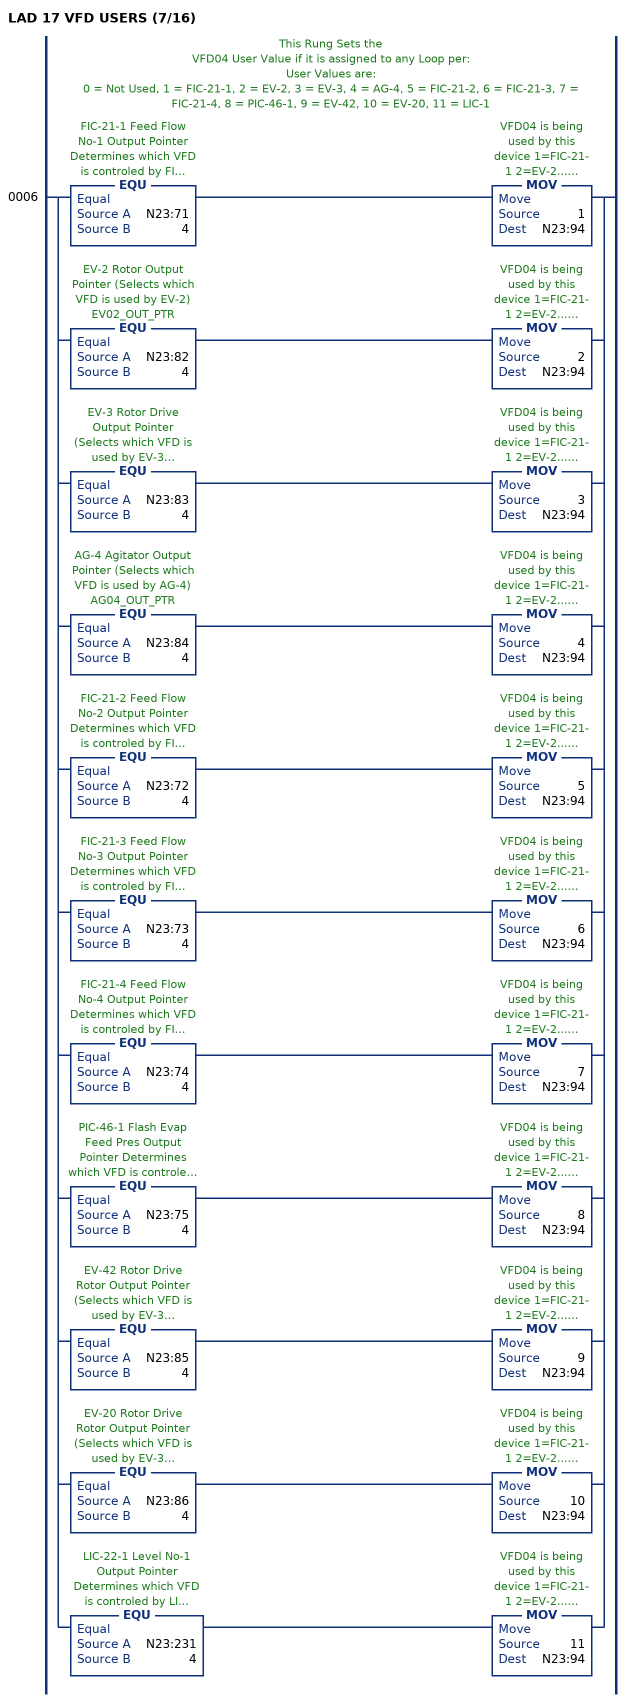
% Rung: 6 %
% This Rung Sets the
% VFD04 User Value if it is assigned to any Loop per:
% 
% User Values are:
% 0 = Not Used, 1 = FIC-21-1, 2 = EV-2, 3 = EV-3, 4 = AG-4, 5 = FIC-21-2, 6 = FIC-21-3, 7 = FIC-21-4, 8 = PIC-46-1, 9 = EV-42, 10 = EV-20, 11 = LIC-1 %
SOR BST EQU N23:71 4 MOV 1 N23:94 NXB EQU N23:82 4 MOV 2 N23:94 NXB EQU N23:83 4 MOV 3 N23:94 NXB EQU N23:84 4 MOV 4 N23:94 NXB EQU N23:72 4 MOV 5 N23:94 NXB EQU N23:73 4 MOV 6 N23:94 NXB EQU N23:74 4 MOV 7 N23:94 NXB EQU N23:75 4 MOV 8 N23:94 NXB EQU N23:85 4 MOV 9 N23:94 NXB EQU N23:86 4 MOV 10 N23:94 NXB EQU N23:231 4 MOV 11 N23:94 BND EOR
%   N23:71  FIC211_OUT_PTR  "FIC-21-1 Feed Flow No-1 Output Pointer Determines which VFD is controled by FIC" %
%   N23:94  VFD04_USER  "VFD04 is being used by this device 1=FIC-21-1 2=EV-2...." %
%   N23:82  EV02_OUT_PTR  "EV-2 Rotor Output Pointer (Selects which VFD is used by EV-2)" %
%   N23:83  EV03_OUT_PTR  "EV-3 Rotor Drive Output Pointer (Selects which VFD is used by EV-3)" %
%   N23:84  AG04_OUT_PTR  "AG-4 Agitator Output Pointer (Selects which VFD is used by AG-4)" %
%   N23:72  FIC212_OUT_PTR  "FIC-21-2 Feed Flow No-2 Output Pointer Determines which VFD is controled by FIC" %
%   N23:73  FIC213_OUT_PTR  "FIC-21-3 Feed Flow No-3 Output Pointer Determines which VFD is controled by FIC" %
%   N23:74  FIC214_OUT_PTR  "FIC-21-4 Feed Flow No-4 Output Pointer Determines which VFD is controled by FIC" %
%   N23:75  PIC461_OUT_PTR  "PIC-46-1 Flash Evap Feed Pres Output Pointer Determines which VFD is controled by FIC" %
%   N23:85  EV42_OUT_PTR  "EV-42 Rotor Drive Rotor Output Pointer (Selects which VFD is used by EV-3)" %
%   N23:86  EV20_OUT_PTR  "EV-20 Rotor Drive Rotor Output Pointer (Selects which VFD is used by EV-3)" %
%   N23:231  LIC221_OUT_PTR  "LIC-22-1 Level No-1 Output Pointer Determines which VFD is controled by LIC" %

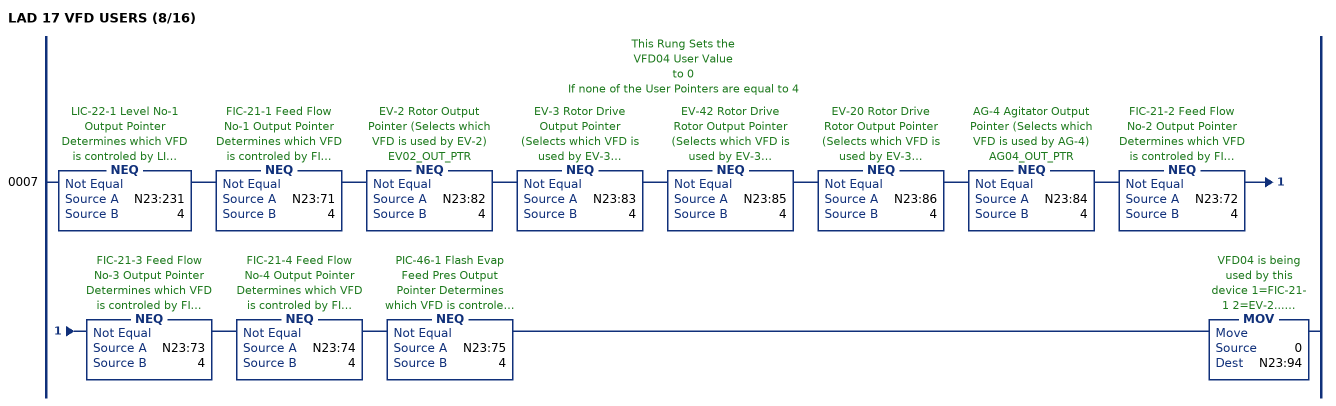
% Rung: 7 %
% This Rung Sets the
% VFD04 User Value
% to 0
% If none of the User Pointers are equal to 4 %
SOR NEQ N23:231 4 NEQ N23:71 4 NEQ N23:82 4 NEQ N23:83 4 NEQ N23:85 4 NEQ N23:86 4 NEQ N23:84 4 NEQ N23:72 4 NEQ N23:73 4 NEQ N23:74 4 NEQ N23:75 4 MOV 0 N23:94 EOR
%   N23:231  LIC221_OUT_PTR  "LIC-22-1 Level No-1 Output Pointer Determines which VFD is controled by LIC" %
%   N23:71  FIC211_OUT_PTR  "FIC-21-1 Feed Flow No-1 Output Pointer Determines which VFD is controled by FIC" %
%   N23:82  EV02_OUT_PTR  "EV-2 Rotor Output Pointer (Selects which VFD is used by EV-2)" %
%   N23:83  EV03_OUT_PTR  "EV-3 Rotor Drive Output Pointer (Selects which VFD is used by EV-3)" %
%   N23:85  EV42_OUT_PTR  "EV-42 Rotor Drive Rotor Output Pointer (Selects which VFD is used by EV-3)" %
%   N23:86  EV20_OUT_PTR  "EV-20 Rotor Drive Rotor Output Pointer (Selects which VFD is used by EV-3)" %
%   N23:84  AG04_OUT_PTR  "AG-4 Agitator Output Pointer (Selects which VFD is used by AG-4)" %
%   N23:72  FIC212_OUT_PTR  "FIC-21-2 Feed Flow No-2 Output Pointer Determines which VFD is controled by FIC" %
%   N23:73  FIC213_OUT_PTR  "FIC-21-3 Feed Flow No-3 Output Pointer Determines which VFD is controled by FIC" %
%   N23:74  FIC214_OUT_PTR  "FIC-21-4 Feed Flow No-4 Output Pointer Determines which VFD is controled by FIC" %
%   N23:75  PIC461_OUT_PTR  "PIC-46-1 Flash Evap Feed Pres Output Pointer Determines which VFD is controled by FIC" %
%   N23:94  VFD04_USER  "VFD04 is being used by this device 1=FIC-21-1 2=EV-2...." %

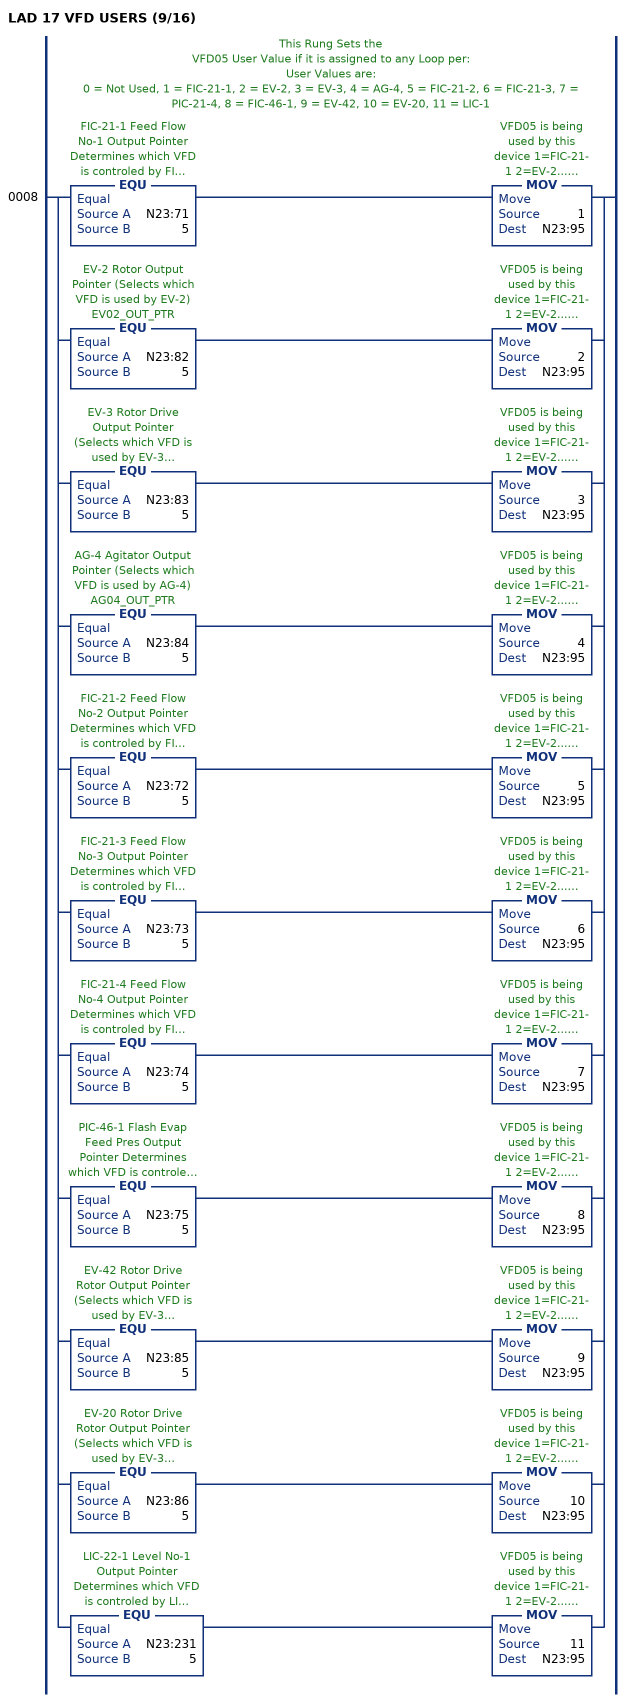
% Rung: 8 %
% This Rung Sets the
% VFD05 User Value if it is assigned to any Loop per:
% 
% User Values are:
% 0 = Not Used, 1 = FIC-21-1, 2 = EV-2, 3 = EV-3, 4 = AG-4, 5 = FIC-21-2, 6 = FIC-21-3, 7 = PIC-21-4, 8 = FIC-46-1, 9 = EV-42, 10 = EV-20, 11 = LIC-1 %
SOR BST EQU N23:71 5 MOV 1 N23:95 NXB EQU N23:82 5 MOV 2 N23:95 NXB EQU N23:83 5 MOV 3 N23:95 NXB EQU N23:84 5 MOV 4 N23:95 NXB EQU N23:72 5 MOV 5 N23:95 NXB EQU N23:73 5 MOV 6 N23:95 NXB EQU N23:74 5 MOV 7 N23:95 NXB EQU N23:75 5 MOV 8 N23:95 NXB EQU N23:85 5 MOV 9 N23:95 NXB EQU N23:86 5 MOV 10 N23:95 NXB EQU N23:231 5 MOV 11 N23:95 BND EOR
%   N23:71  FIC211_OUT_PTR  "FIC-21-1 Feed Flow No-1 Output Pointer Determines which VFD is controled by FIC" %
%   N23:95  VFD05_USER  "VFD05 is being used by this device 1=FIC-21-1 2=EV-2...." %
%   N23:82  EV02_OUT_PTR  "EV-2 Rotor Output Pointer (Selects which VFD is used by EV-2)" %
%   N23:83  EV03_OUT_PTR  "EV-3 Rotor Drive Output Pointer (Selects which VFD is used by EV-3)" %
%   N23:84  AG04_OUT_PTR  "AG-4 Agitator Output Pointer (Selects which VFD is used by AG-4)" %
%   N23:72  FIC212_OUT_PTR  "FIC-21-2 Feed Flow No-2 Output Pointer Determines which VFD is controled by FIC" %
%   N23:73  FIC213_OUT_PTR  "FIC-21-3 Feed Flow No-3 Output Pointer Determines which VFD is controled by FIC" %
%   N23:74  FIC214_OUT_PTR  "FIC-21-4 Feed Flow No-4 Output Pointer Determines which VFD is controled by FIC" %
%   N23:75  PIC461_OUT_PTR  "PIC-46-1 Flash Evap Feed Pres Output Pointer Determines which VFD is controled by FIC" %
%   N23:85  EV42_OUT_PTR  "EV-42 Rotor Drive Rotor Output Pointer (Selects which VFD is used by EV-3)" %
%   N23:86  EV20_OUT_PTR  "EV-20 Rotor Drive Rotor Output Pointer (Selects which VFD is used by EV-3)" %
%   N23:231  LIC221_OUT_PTR  "LIC-22-1 Level No-1 Output Pointer Determines which VFD is controled by LIC" %

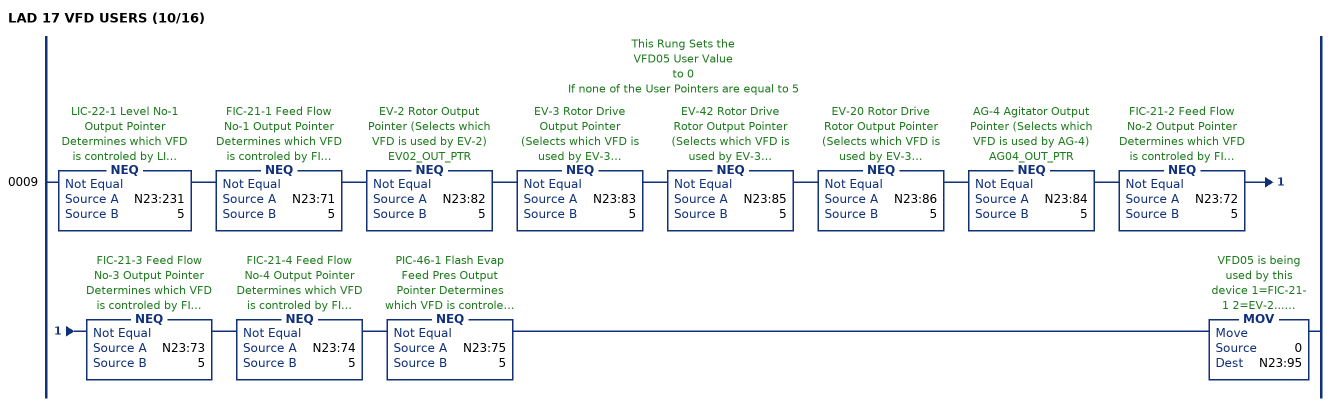
% Rung: 9 %
% This Rung Sets the
% VFD05 User Value
% to 0
% If none of the User Pointers are equal to 5 %
SOR NEQ N23:231 5 NEQ N23:71 5 NEQ N23:82 5 NEQ N23:83 5 NEQ N23:85 5 NEQ N23:86 5 NEQ N23:84 5 NEQ N23:72 5 NEQ N23:73 5 NEQ N23:74 5 NEQ N23:75 5 MOV 0 N23:95 EOR
%   N23:231  LIC221_OUT_PTR  "LIC-22-1 Level No-1 Output Pointer Determines which VFD is controled by LIC" %
%   N23:71  FIC211_OUT_PTR  "FIC-21-1 Feed Flow No-1 Output Pointer Determines which VFD is controled by FIC" %
%   N23:82  EV02_OUT_PTR  "EV-2 Rotor Output Pointer (Selects which VFD is used by EV-2)" %
%   N23:83  EV03_OUT_PTR  "EV-3 Rotor Drive Output Pointer (Selects which VFD is used by EV-3)" %
%   N23:85  EV42_OUT_PTR  "EV-42 Rotor Drive Rotor Output Pointer (Selects which VFD is used by EV-3)" %
%   N23:86  EV20_OUT_PTR  "EV-20 Rotor Drive Rotor Output Pointer (Selects which VFD is used by EV-3)" %
%   N23:84  AG04_OUT_PTR  "AG-4 Agitator Output Pointer (Selects which VFD is used by AG-4)" %
%   N23:72  FIC212_OUT_PTR  "FIC-21-2 Feed Flow No-2 Output Pointer Determines which VFD is controled by FIC" %
%   N23:73  FIC213_OUT_PTR  "FIC-21-3 Feed Flow No-3 Output Pointer Determines which VFD is controled by FIC" %
%   N23:74  FIC214_OUT_PTR  "FIC-21-4 Feed Flow No-4 Output Pointer Determines which VFD is controled by FIC" %
%   N23:75  PIC461_OUT_PTR  "PIC-46-1 Flash Evap Feed Pres Output Pointer Determines which VFD is controled by FIC" %
%   N23:95  VFD05_USER  "VFD05 is being used by this device 1=FIC-21-1 2=EV-2...." %

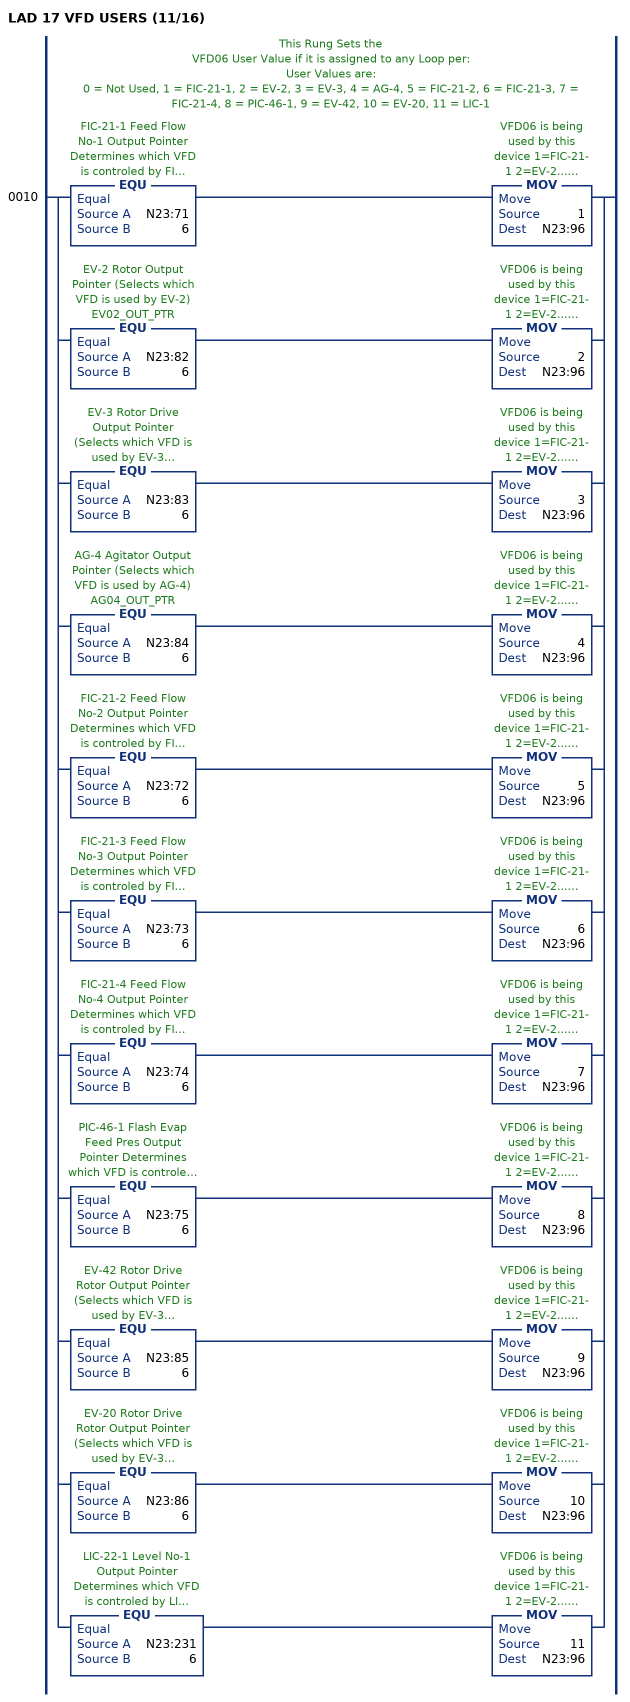
% Rung: 10 %
% This Rung Sets the
% VFD06 User Value if it is assigned to any Loop per:
% 
% User Values are:
% 0 = Not Used, 1 = FIC-21-1, 2 = EV-2, 3 = EV-3, 4 = AG-4, 5 = FIC-21-2, 6 = FIC-21-3, 7 = FIC-21-4, 8 = PIC-46-1, 9 = EV-42, 10 = EV-20, 11 = LIC-1 %
SOR BST EQU N23:71 6 MOV 1 N23:96 NXB EQU N23:82 6 MOV 2 N23:96 NXB EQU N23:83 6 MOV 3 N23:96 NXB EQU N23:84 6 MOV 4 N23:96 NXB EQU N23:72 6 MOV 5 N23:96 NXB EQU N23:73 6 MOV 6 N23:96 NXB EQU N23:74 6 MOV 7 N23:96 NXB EQU N23:75 6 MOV 8 N23:96 NXB EQU N23:85 6 MOV 9 N23:96 NXB EQU N23:86 6 MOV 10 N23:96 NXB EQU N23:231 6 MOV 11 N23:96 BND EOR
%   N23:71  FIC211_OUT_PTR  "FIC-21-1 Feed Flow No-1 Output Pointer Determines which VFD is controled by FIC" %
%   N23:96  VFD06_USER  "VFD06 is being used by this device 1=FIC-21-1 2=EV-2...." %
%   N23:82  EV02_OUT_PTR  "EV-2 Rotor Output Pointer (Selects which VFD is used by EV-2)" %
%   N23:83  EV03_OUT_PTR  "EV-3 Rotor Drive Output Pointer (Selects which VFD is used by EV-3)" %
%   N23:84  AG04_OUT_PTR  "AG-4 Agitator Output Pointer (Selects which VFD is used by AG-4)" %
%   N23:72  FIC212_OUT_PTR  "FIC-21-2 Feed Flow No-2 Output Pointer Determines which VFD is controled by FIC" %
%   N23:73  FIC213_OUT_PTR  "FIC-21-3 Feed Flow No-3 Output Pointer Determines which VFD is controled by FIC" %
%   N23:74  FIC214_OUT_PTR  "FIC-21-4 Feed Flow No-4 Output Pointer Determines which VFD is controled by FIC" %
%   N23:75  PIC461_OUT_PTR  "PIC-46-1 Flash Evap Feed Pres Output Pointer Determines which VFD is controled by FIC" %
%   N23:85  EV42_OUT_PTR  "EV-42 Rotor Drive Rotor Output Pointer (Selects which VFD is used by EV-3)" %
%   N23:86  EV20_OUT_PTR  "EV-20 Rotor Drive Rotor Output Pointer (Selects which VFD is used by EV-3)" %
%   N23:231  LIC221_OUT_PTR  "LIC-22-1 Level No-1 Output Pointer Determines which VFD is controled by LIC" %

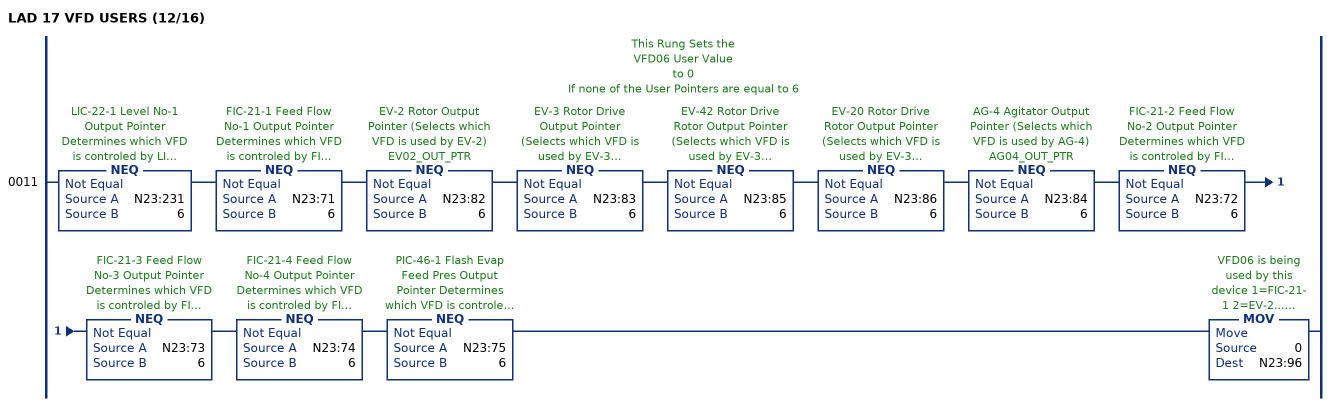
% Rung: 11 %
% This Rung Sets the
% VFD06 User Value
% to 0
% If none of the User Pointers are equal to 6 %
SOR NEQ N23:231 6 NEQ N23:71 6 NEQ N23:82 6 NEQ N23:83 6 NEQ N23:85 6 NEQ N23:86 6 NEQ N23:84 6 NEQ N23:72 6 NEQ N23:73 6 NEQ N23:74 6 NEQ N23:75 6 MOV 0 N23:96 EOR
%   N23:231  LIC221_OUT_PTR  "LIC-22-1 Level No-1 Output Pointer Determines which VFD is controled by LIC" %
%   N23:71  FIC211_OUT_PTR  "FIC-21-1 Feed Flow No-1 Output Pointer Determines which VFD is controled by FIC" %
%   N23:82  EV02_OUT_PTR  "EV-2 Rotor Output Pointer (Selects which VFD is used by EV-2)" %
%   N23:83  EV03_OUT_PTR  "EV-3 Rotor Drive Output Pointer (Selects which VFD is used by EV-3)" %
%   N23:85  EV42_OUT_PTR  "EV-42 Rotor Drive Rotor Output Pointer (Selects which VFD is used by EV-3)" %
%   N23:86  EV20_OUT_PTR  "EV-20 Rotor Drive Rotor Output Pointer (Selects which VFD is used by EV-3)" %
%   N23:84  AG04_OUT_PTR  "AG-4 Agitator Output Pointer (Selects which VFD is used by AG-4)" %
%   N23:72  FIC212_OUT_PTR  "FIC-21-2 Feed Flow No-2 Output Pointer Determines which VFD is controled by FIC" %
%   N23:73  FIC213_OUT_PTR  "FIC-21-3 Feed Flow No-3 Output Pointer Determines which VFD is controled by FIC" %
%   N23:74  FIC214_OUT_PTR  "FIC-21-4 Feed Flow No-4 Output Pointer Determines which VFD is controled by FIC" %
%   N23:75  PIC461_OUT_PTR  "PIC-46-1 Flash Evap Feed Pres Output Pointer Determines which VFD is controled by FIC" %
%   N23:96  VFD06_USER  "VFD06 is being used by this device 1=FIC-21-1 2=EV-2...." %

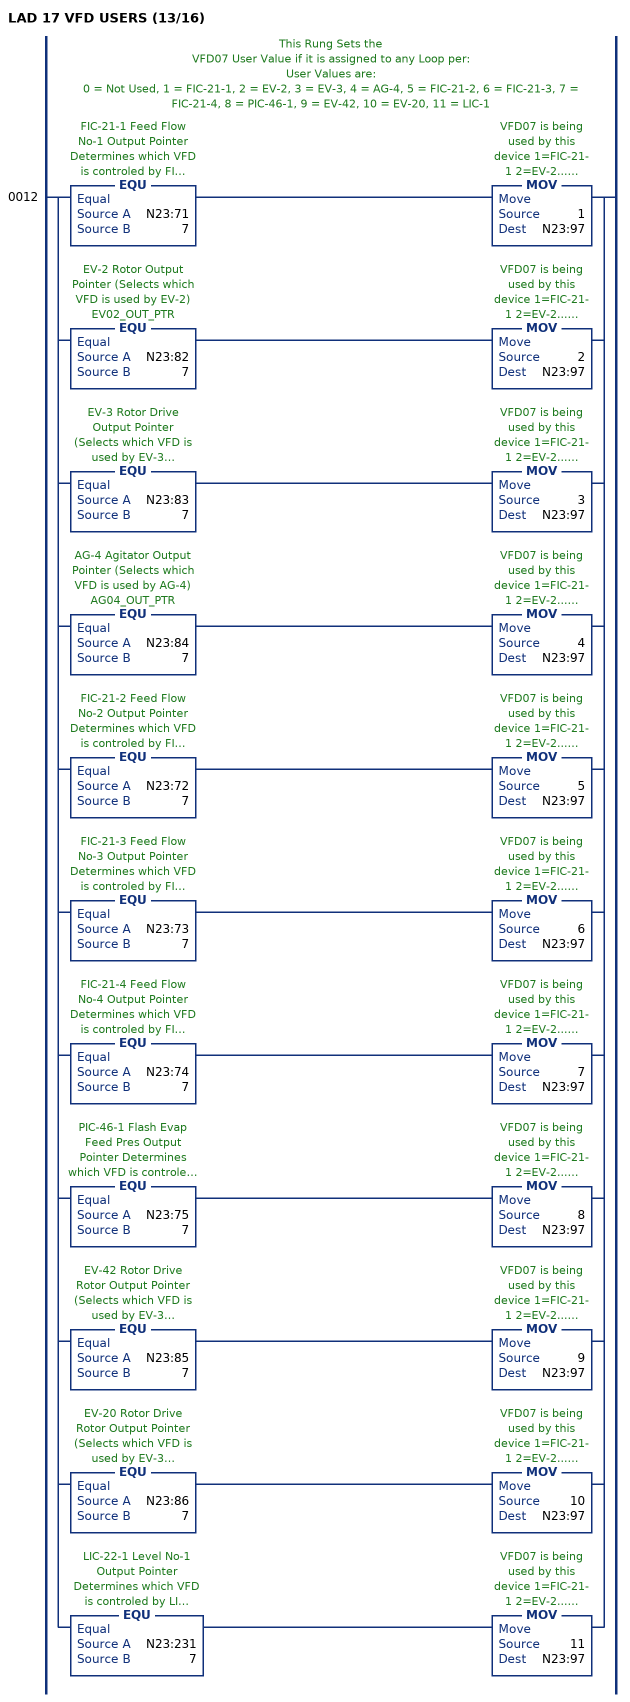
% Rung: 12 %
% This Rung Sets the
% VFD07 User Value if it is assigned to any Loop per:
% 
% User Values are:
% 0 = Not Used, 1 = FIC-21-1, 2 = EV-2, 3 = EV-3, 4 = AG-4, 5 = FIC-21-2, 6 = FIC-21-3, 7 = FIC-21-4, 8 = PIC-46-1, 9 = EV-42, 10 = EV-20, 11 = LIC-1 %
SOR BST EQU N23:71 7 MOV 1 N23:97 NXB EQU N23:82 7 MOV 2 N23:97 NXB EQU N23:83 7 MOV 3 N23:97 NXB EQU N23:84 7 MOV 4 N23:97 NXB EQU N23:72 7 MOV 5 N23:97 NXB EQU N23:73 7 MOV 6 N23:97 NXB EQU N23:74 7 MOV 7 N23:97 NXB EQU N23:75 7 MOV 8 N23:97 NXB EQU N23:85 7 MOV 9 N23:97 NXB EQU N23:86 7 MOV 10 N23:97 NXB EQU N23:231 7 MOV 11 N23:97 BND EOR
%   N23:71  FIC211_OUT_PTR  "FIC-21-1 Feed Flow No-1 Output Pointer Determines which VFD is controled by FIC" %
%   N23:97  VFD07_USER  "VFD07 is being used by this device 1=FIC-21-1 2=EV-2...." %
%   N23:82  EV02_OUT_PTR  "EV-2 Rotor Output Pointer (Selects which VFD is used by EV-2)" %
%   N23:83  EV03_OUT_PTR  "EV-3 Rotor Drive Output Pointer (Selects which VFD is used by EV-3)" %
%   N23:84  AG04_OUT_PTR  "AG-4 Agitator Output Pointer (Selects which VFD is used by AG-4)" %
%   N23:72  FIC212_OUT_PTR  "FIC-21-2 Feed Flow No-2 Output Pointer Determines which VFD is controled by FIC" %
%   N23:73  FIC213_OUT_PTR  "FIC-21-3 Feed Flow No-3 Output Pointer Determines which VFD is controled by FIC" %
%   N23:74  FIC214_OUT_PTR  "FIC-21-4 Feed Flow No-4 Output Pointer Determines which VFD is controled by FIC" %
%   N23:75  PIC461_OUT_PTR  "PIC-46-1 Flash Evap Feed Pres Output Pointer Determines which VFD is controled by FIC" %
%   N23:85  EV42_OUT_PTR  "EV-42 Rotor Drive Rotor Output Pointer (Selects which VFD is used by EV-3)" %
%   N23:86  EV20_OUT_PTR  "EV-20 Rotor Drive Rotor Output Pointer (Selects which VFD is used by EV-3)" %
%   N23:231  LIC221_OUT_PTR  "LIC-22-1 Level No-1 Output Pointer Determines which VFD is controled by LIC" %

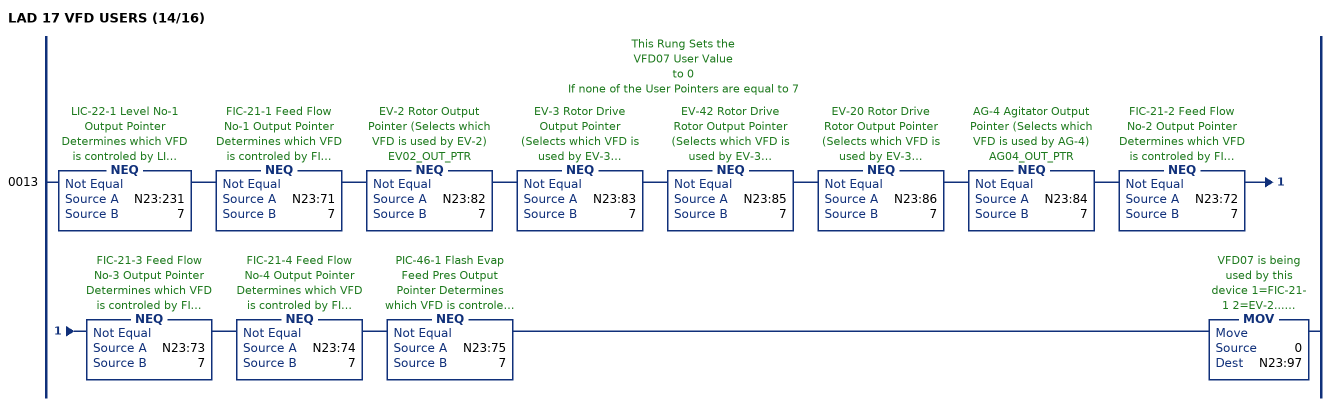
% Rung: 13 %
% This Rung Sets the
% VFD07 User Value
% to 0
% If none of the User Pointers are equal to 7 %
SOR NEQ N23:231 7 NEQ N23:71 7 NEQ N23:82 7 NEQ N23:83 7 NEQ N23:85 7 NEQ N23:86 7 NEQ N23:84 7 NEQ N23:72 7 NEQ N23:73 7 NEQ N23:74 7 NEQ N23:75 7 MOV 0 N23:97 EOR
%   N23:231  LIC221_OUT_PTR  "LIC-22-1 Level No-1 Output Pointer Determines which VFD is controled by LIC" %
%   N23:71  FIC211_OUT_PTR  "FIC-21-1 Feed Flow No-1 Output Pointer Determines which VFD is controled by FIC" %
%   N23:82  EV02_OUT_PTR  "EV-2 Rotor Output Pointer (Selects which VFD is used by EV-2)" %
%   N23:83  EV03_OUT_PTR  "EV-3 Rotor Drive Output Pointer (Selects which VFD is used by EV-3)" %
%   N23:85  EV42_OUT_PTR  "EV-42 Rotor Drive Rotor Output Pointer (Selects which VFD is used by EV-3)" %
%   N23:86  EV20_OUT_PTR  "EV-20 Rotor Drive Rotor Output Pointer (Selects which VFD is used by EV-3)" %
%   N23:84  AG04_OUT_PTR  "AG-4 Agitator Output Pointer (Selects which VFD is used by AG-4)" %
%   N23:72  FIC212_OUT_PTR  "FIC-21-2 Feed Flow No-2 Output Pointer Determines which VFD is controled by FIC" %
%   N23:73  FIC213_OUT_PTR  "FIC-21-3 Feed Flow No-3 Output Pointer Determines which VFD is controled by FIC" %
%   N23:74  FIC214_OUT_PTR  "FIC-21-4 Feed Flow No-4 Output Pointer Determines which VFD is controled by FIC" %
%   N23:75  PIC461_OUT_PTR  "PIC-46-1 Flash Evap Feed Pres Output Pointer Determines which VFD is controled by FIC" %
%   N23:97  VFD07_USER  "VFD07 is being used by this device 1=FIC-21-1 2=EV-2...." %

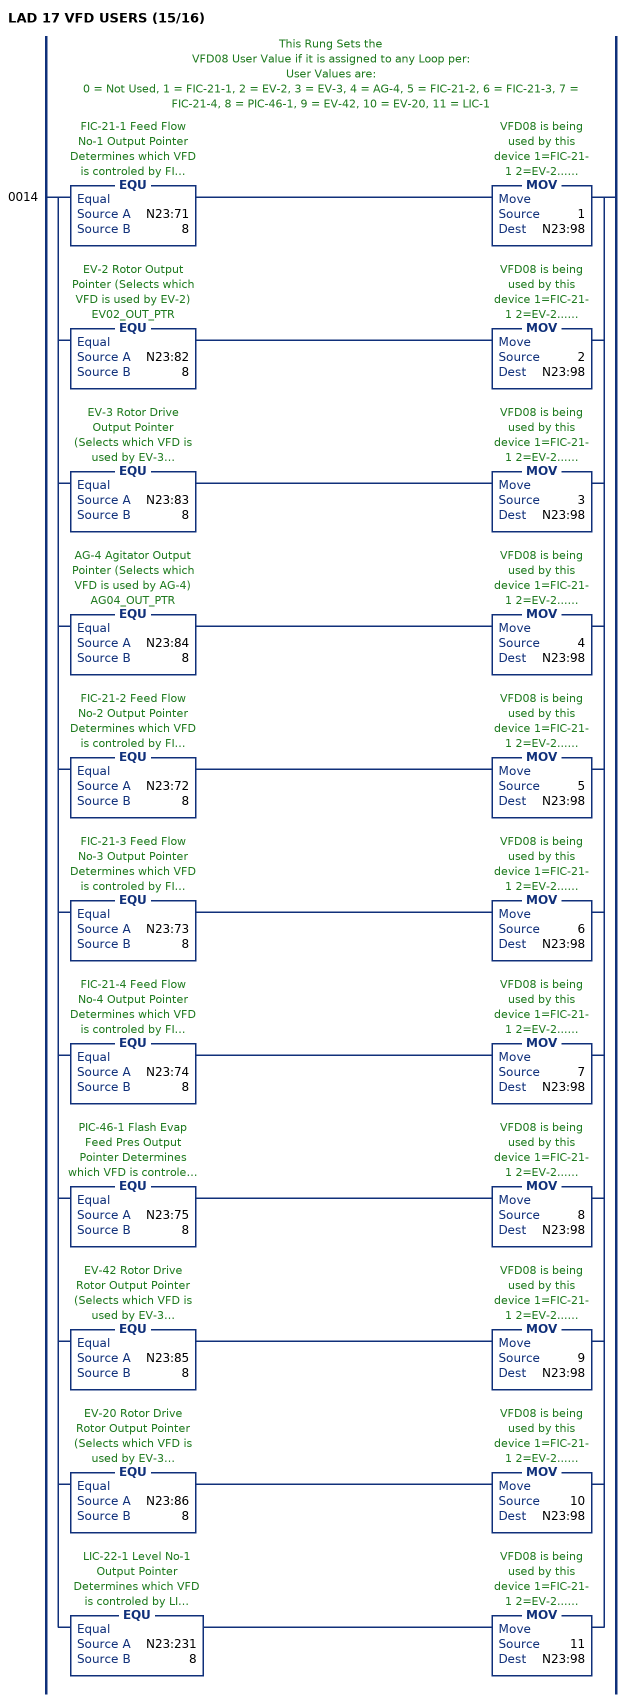
% Rung: 14 %
% This Rung Sets the
% VFD08 User Value if it is assigned to any Loop per:
% 
% User Values are:
% 0 = Not Used, 1 = FIC-21-1, 2 = EV-2, 3 = EV-3, 4 = AG-4, 5 = FIC-21-2, 6 = FIC-21-3, 7 = FIC-21-4, 8 = PIC-46-1, 9 = EV-42, 10 = EV-20, 11 = LIC-1 %
SOR BST EQU N23:71 8 MOV 1 N23:98 NXB EQU N23:82 8 MOV 2 N23:98 NXB EQU N23:83 8 MOV 3 N23:98 NXB EQU N23:84 8 MOV 4 N23:98 NXB EQU N23:72 8 MOV 5 N23:98 NXB EQU N23:73 8 MOV 6 N23:98 NXB EQU N23:74 8 MOV 7 N23:98 NXB EQU N23:75 8 MOV 8 N23:98 NXB EQU N23:85 8 MOV 9 N23:98 NXB EQU N23:86 8 MOV 10 N23:98 NXB EQU N23:231 8 MOV 11 N23:98 BND EOR
%   N23:71  FIC211_OUT_PTR  "FIC-21-1 Feed Flow No-1 Output Pointer Determines which VFD is controled by FIC" %
%   N23:98  VFD08_USER  "VFD08 is being used by this device 1=FIC-21-1 2=EV-2...." %
%   N23:82  EV02_OUT_PTR  "EV-2 Rotor Output Pointer (Selects which VFD is used by EV-2)" %
%   N23:83  EV03_OUT_PTR  "EV-3 Rotor Drive Output Pointer (Selects which VFD is used by EV-3)" %
%   N23:84  AG04_OUT_PTR  "AG-4 Agitator Output Pointer (Selects which VFD is used by AG-4)" %
%   N23:72  FIC212_OUT_PTR  "FIC-21-2 Feed Flow No-2 Output Pointer Determines which VFD is controled by FIC" %
%   N23:73  FIC213_OUT_PTR  "FIC-21-3 Feed Flow No-3 Output Pointer Determines which VFD is controled by FIC" %
%   N23:74  FIC214_OUT_PTR  "FIC-21-4 Feed Flow No-4 Output Pointer Determines which VFD is controled by FIC" %
%   N23:75  PIC461_OUT_PTR  "PIC-46-1 Flash Evap Feed Pres Output Pointer Determines which VFD is controled by FIC" %
%   N23:85  EV42_OUT_PTR  "EV-42 Rotor Drive Rotor Output Pointer (Selects which VFD is used by EV-3)" %
%   N23:86  EV20_OUT_PTR  "EV-20 Rotor Drive Rotor Output Pointer (Selects which VFD is used by EV-3)" %
%   N23:231  LIC221_OUT_PTR  "LIC-22-1 Level No-1 Output Pointer Determines which VFD is controled by LIC" %

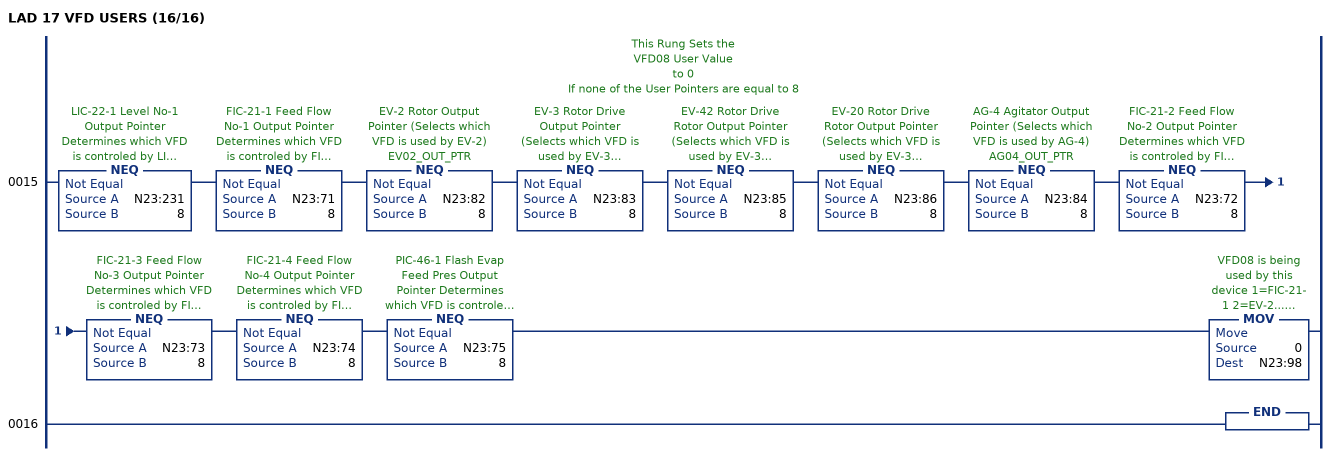
% Rung: 15 %
% This Rung Sets the
% VFD08 User Value
% to 0
% If none of the User Pointers are equal to 8 %
SOR NEQ N23:231 8 NEQ N23:71 8 NEQ N23:82 8 NEQ N23:83 8 NEQ N23:85 8 NEQ N23:86 8 NEQ N23:84 8 NEQ N23:72 8 NEQ N23:73 8 NEQ N23:74 8 NEQ N23:75 8 MOV 0 N23:98 EOR
%   N23:231  LIC221_OUT_PTR  "LIC-22-1 Level No-1 Output Pointer Determines which VFD is controled by LIC" %
%   N23:71  FIC211_OUT_PTR  "FIC-21-1 Feed Flow No-1 Output Pointer Determines which VFD is controled by FIC" %
%   N23:82  EV02_OUT_PTR  "EV-2 Rotor Output Pointer (Selects which VFD is used by EV-2)" %
%   N23:83  EV03_OUT_PTR  "EV-3 Rotor Drive Output Pointer (Selects which VFD is used by EV-3)" %
%   N23:85  EV42_OUT_PTR  "EV-42 Rotor Drive Rotor Output Pointer (Selects which VFD is used by EV-3)" %
%   N23:86  EV20_OUT_PTR  "EV-20 Rotor Drive Rotor Output Pointer (Selects which VFD is used by EV-3)" %
%   N23:84  AG04_OUT_PTR  "AG-4 Agitator Output Pointer (Selects which VFD is used by AG-4)" %
%   N23:72  FIC212_OUT_PTR  "FIC-21-2 Feed Flow No-2 Output Pointer Determines which VFD is controled by FIC" %
%   N23:73  FIC213_OUT_PTR  "FIC-21-3 Feed Flow No-3 Output Pointer Determines which VFD is controled by FIC" %
%   N23:74  FIC214_OUT_PTR  "FIC-21-4 Feed Flow No-4 Output Pointer Determines which VFD is controled by FIC" %
%   N23:75  PIC461_OUT_PTR  "PIC-46-1 Flash Evap Feed Pres Output Pointer Determines which VFD is controled by FIC" %
%   N23:98  VFD08_USER  "VFD08 is being used by this device 1=FIC-21-1 2=EV-2...." %
% Rung: 16 %
SOR END EOR

LADDER 31 "MOVE TES"    % Move TE Info to Sequencial Locations, etc %
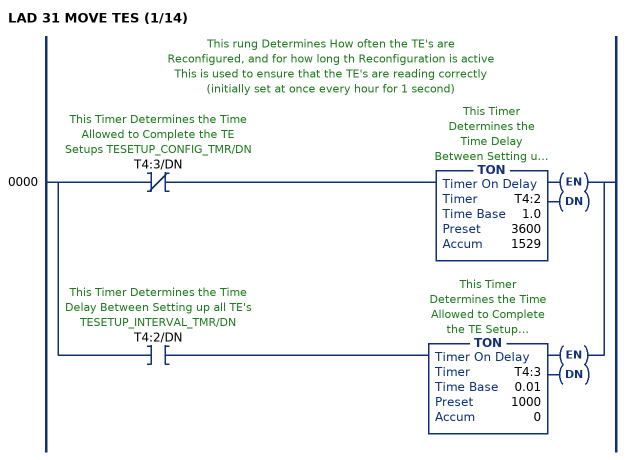
% Rung: 0 %
% This rung Determines How often the TE's are
% Reconfigured, and for how long th Reconfiguration is active
% This is used to ensure that the TE's are reading correctly
%    (initially set at once every hour for 1 second) %
SOR BST XIO T4:3/DN TON T4:2 1.0 3600 1529 NXB XIC T4:2/DN TON T4:3 0.01 1000 0 BND EOR
%   T4:3  TESETUP_CONFIG_TMR  "This Timer Determines the Time Allowed to Complete the TE Setups" %
%   T4:2  TESETUP_INTERVAL_TMR  "This Timer Determines the Time Delay Between Setting up all TE's" %

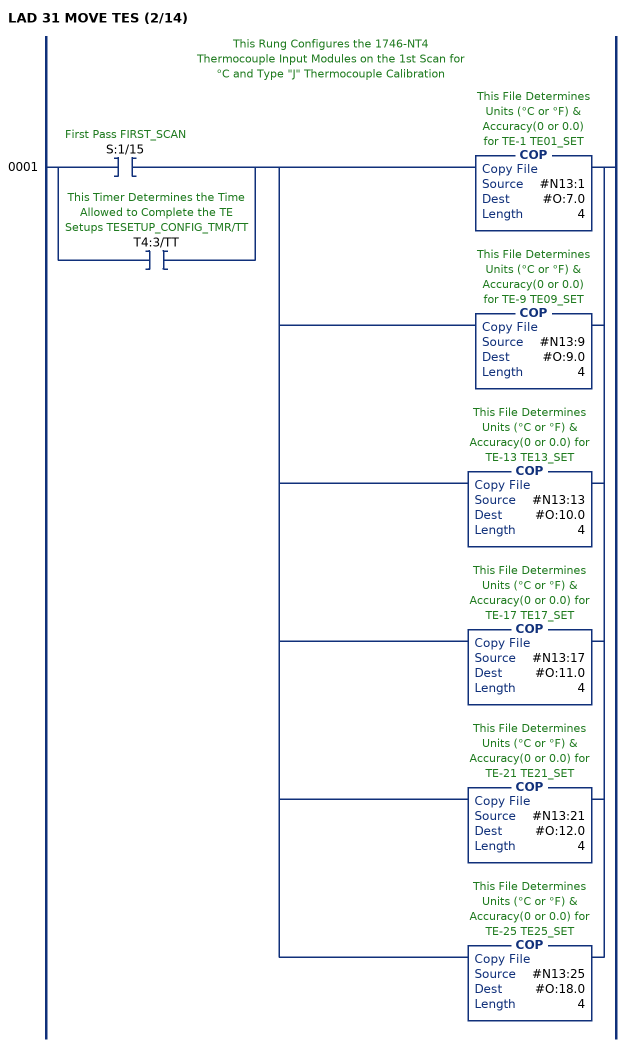
% Rung: 1 %
% This Rung Configures the 1746-NT4
% Thermocouple Input Modules on the 1st Scan for
% °C and Type "J" Thermocouple Calibration %
SOR BST XIC S:1/15 NXB XIC T4:3/TT BND BST COP #N13:1 #O:7.0 4 NXB COP #N13:9 #O:9.0 4 NXB COP #N13:13 #O:10.0 4 NXB COP #N13:17 #O:11.0 4 NXB COP #N13:21 #O:12.0 4 NXB COP #N13:25 #O:18.0 4 BND EOR
%   S:1/15  FIRST_SCAN  "First Pass" %
%   T4:3  TESETUP_CONFIG_TMR  "This Timer Determines the Time Allowed to Complete the TE Setups" %
%   N13:1  TE01_SETUP  "This File Determines Units (°C or °F) & Accuracy(0 or 0.0) for TE-1" %
%   O:7.0  TE01_SET  "This File Determines Units (°C or °F) & Accuracy(0 or 0.0) for TE-1" %
%   N13:9  TE09_SETUP  "This File Determines Units (°C or °F) & Accuracy(0 or 0.0) for TE-9" %
%   O:9.0  TE09_SET  "This File Determines Units (°C or °F) & Accuracy(0 or 0.0) for TE-9" %
%   N13:13  TE13_SETUP  "This File Determines Units (°C or °F) & Accuracy(0 or 0.0) for TE-13" %
%   O:10.0  TE13_SET  "This File Determines Units (°C or °F) & Accuracy(0 or 0.0) for TE-13" %
%   N13:17  TE17_SETUP  "This File Determines Units (°C or °F) & Accuracy(0 or 0.0) for TE-17" %
%   O:11.0  TE17_SET  "This File Determines Units (°C or °F) & Accuracy(0 or 0.0) for TE-17" %
%   N13:21  TE21_SETUP  "This File Determines Units (°C or °F) & Accuracy(0 or 0.0) for TE-21" %
%   O:12.0  TE21_SET  "This File Determines Units (°C or °F) & Accuracy(0 or 0.0) for TE-21" %
%   N13:25  TE25_SETUP  "This File Determines Units (°C or °F) & Accuracy(0 or 0.0) for TE-25" %
%   O:18.0  TE25_SET  "This File Determines Units (°C or °F) & Accuracy(0 or 0.0) for TE-25" %

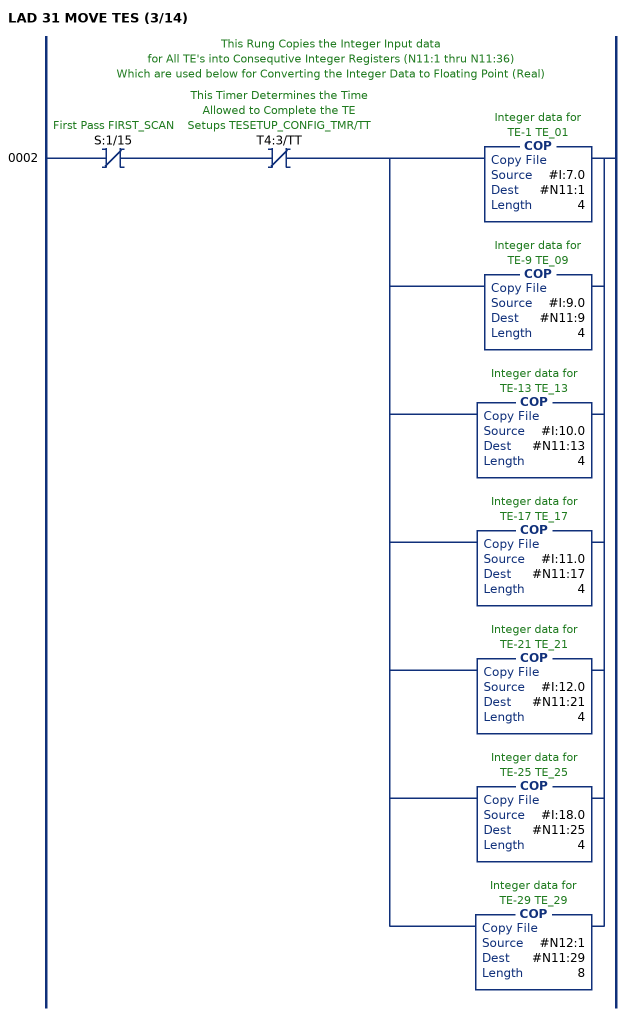
% Rung: 2 %
% This Rung Copies the Integer Input data
% for All TE's into Consequtive Integer Registers (N11:1 thru N11:36)
% Which are used below for Converting the Integer Data to Floating Point (Real) %
SOR XIO S:1/15 XIO T4:3/TT BST COP #I:7.0 #N11:1 4 NXB COP #I:9.0 #N11:9 4 NXB COP #I:10.0 #N11:13 4 NXB COP #I:11.0 #N11:17 4 NXB COP #I:12.0 #N11:21 4 NXB COP #I:18.0 #N11:25 4 NXB COP #N12:1 #N11:29 8 BND EOR
%   S:1/15  FIRST_SCAN  "First Pass" %
%   T4:3  TESETUP_CONFIG_TMR  "This Timer Determines the Time Allowed to Complete the TE Setups" %
%   I:7.0  TE01_BIN  "Binary Input data for TE-1" %
%   N11:1  TE_01  "Integer data for TE-1" %
%   I:9.0  TE09_BIN  "Binary Input data for TE-9" %
%   N11:9  TE_09  "Integer data for TE-9" %
%   I:10.0  TE13_BIN  "Binary Input data for TE-13" %
%   N11:13  TE_13  "Integer data for TE-13" %
%   I:11.0  TE17_BIN  "Binary Input data for TE-17" %
%   N11:17  TE_17  "Integer data for TE-17" %
%   I:12.0  TE21_BIN  "Binary Input data for TE-21" %
%   N11:21  TE_21  "Integer data for TE-21" %
%   I:18.0  TE25_BIN  "Binary Input data for TE-25" %
%   N11:25  TE_25  "Integer data for TE-25" %
%   N12:1  TE29_BIN  "Binary data for TE-29" %
%   N11:29  TE_29  "Integer data for TE-29" %

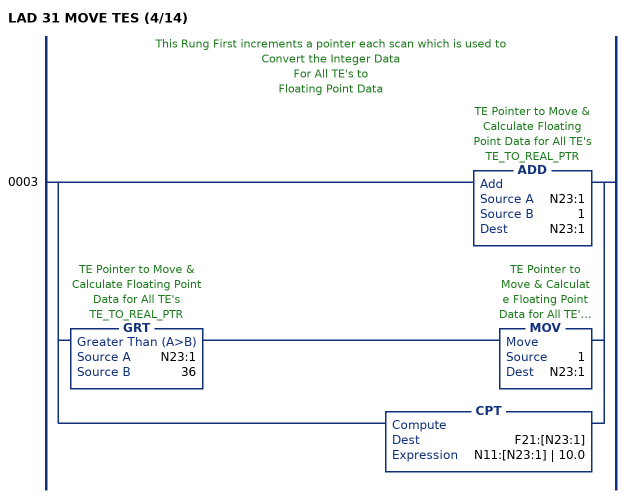
% Rung: 3 %
% This Rung First increments a pointer each scan which is used to
% Convert the Integer Data
% For All TE's to
% Floating Point Data %
SOR BST ADD N23:1 1 N23:1 NXB GRT N23:1 36 MOV 1 N23:1 NXB CPT F21:[N23:1] " N11:[N23:1] | 10.0 " BND EOR
%   N23:1  TE_TO_REAL_PTR  "TE Pointer to Move & Calculate Floating Point Data for All TE's" %

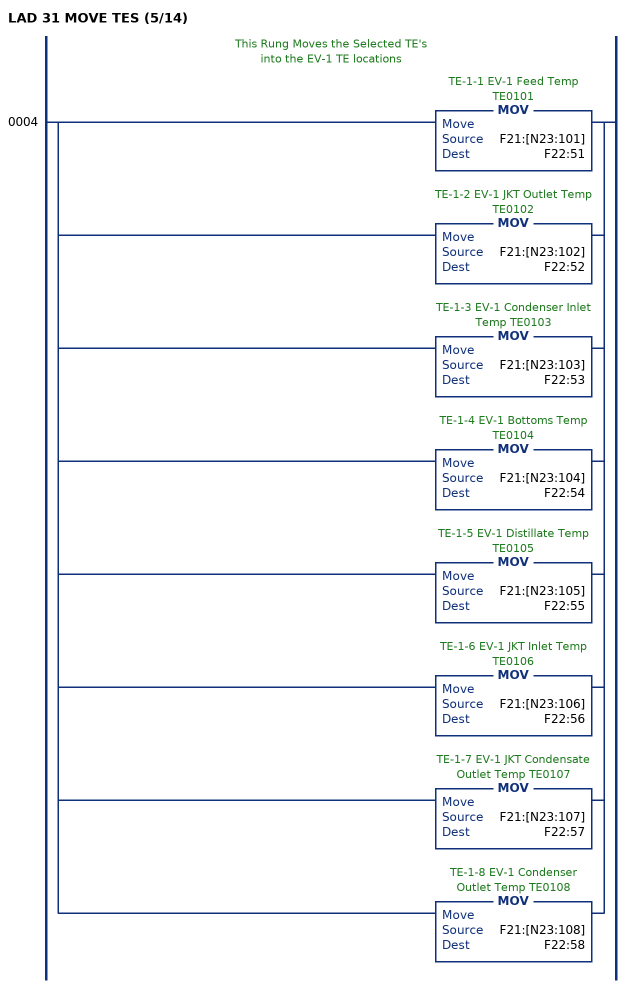
% Rung: 4 %
% This Rung Moves the Selected TE's
% into the EV-1 TE locations %
SOR BST MOV F21:[N23:101] F22:51 NXB MOV F21:[N23:102] F22:52 NXB MOV F21:[N23:103] F22:53 NXB MOV F21:[N23:104] F22:54 NXB MOV F21:[N23:105] F22:55 NXB MOV F21:[N23:106] F22:56 NXB MOV F21:[N23:107] F22:57 NXB MOV F21:[N23:108] F22:58 BND EOR
%   N23:101  TE0101_PTR  "TE-1-1 Pointer" %
%   F22:51  TE0101  "TE-1-1 EV-1 Feed Temp" %
%   N23:102  TE0102_PTR  "TE-1-2 Pointer" %
%   F22:52  TE0102  "TE-1-2 EV-1 JKT Outlet Temp" %
%   N23:103  TE0103_PTR  "TE-1-3 Pointer" %
%   F22:53  TE0103  "TE-1-3 EV-1 Condenser Inlet Temp" %
%   N23:104  TE0104_PTR  "TE-1-4 Pointer" %
%   F22:54  TE0104  "TE-1-4 EV-1 Bottoms Temp" %
%   N23:105  TE0105_PTR  "TE-1-5 Pointer" %
%   F22:55  TE0105  "TE-1-5 EV-1 Distillate Temp" %
%   N23:106  TE0106_PTR  "TE-1-6 Pointer" %
%   F22:56  TE0106  "TE-1-6 EV-1 JKT Inlet Temp" %
%   N23:107  TE0107_PTR  "TE-1-7 Pointer" %
%   F22:57  TE0107  "TE-1-7 EV-1 JKT Condensate Outlet Temp" %
%   N23:108  TE0108_PTR  "TE-1-8 Pointer" %
%   F22:58  TE0108  "TE-1-8 EV-1 Condenser Outlet Temp" %

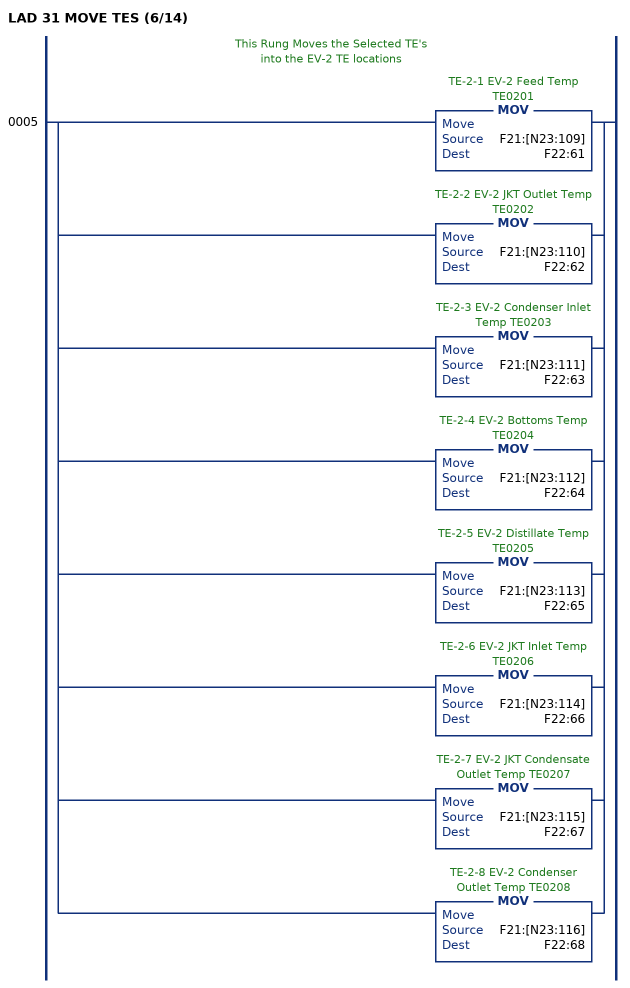
% Rung: 5 %
% This Rung Moves the Selected TE's
% into the EV-2 TE locations %
SOR BST MOV F21:[N23:109] F22:61 NXB MOV F21:[N23:110] F22:62 NXB MOV F21:[N23:111] F22:63 NXB MOV F21:[N23:112] F22:64 NXB MOV F21:[N23:113] F22:65 NXB MOV F21:[N23:114] F22:66 NXB MOV F21:[N23:115] F22:67 NXB MOV F21:[N23:116] F22:68 BND EOR
%   N23:109  TE0201_PTR  "TE-2-1 EV-2 Feed Temp PTR" %
%   F22:61  TE0201  "TE-2-1 EV-2 Feed Temp" %
%   N23:110  TE0202_PTR  "TE-2-2 EV-2 JKT Outlet Temp PTR" %
%   F22:62  TE0202  "TE-2-2 EV-2 JKT Outlet Temp" %
%   N23:111  TE0203_PTR  "TE-2-3 EV-2 Condenser Inlet Temp PTR" %
%   F22:63  TE0203  "TE-2-3 EV-2 Condenser Inlet Temp" %
%   N23:112  TE0204_PTR  "TE-2-4 EV-2 Bottoms Temp PTR" %
%   F22:64  TE0204  "TE-2-4 EV-2 Bottoms Temp" %
%   N23:113  TE0205_PTR  "TE-2-5 EV-2 Distillate Temp PTR" %
%   F22:65  TE0205  "TE-2-5 EV-2 Distillate Temp" %
%   N23:114  TE0206_PTR  "TE-2-6 EV-2 JKT Inlet Temp PTR" %
%   F22:66  TE0206  "TE-2-6 EV-2 JKT Inlet Temp" %
%   N23:115  TE0207_PTR  "TE-2-7 EV-2 JKT Condensate Outlet Temp PTR" %
%   F22:67  TE0207  "TE-2-7 EV-2 JKT Condensate Outlet Temp" %
%   N23:116  TE0208_PTR  "TE-2-8 EV-2 Condenser Outlet Temp PTR" %
%   F22:68  TE0208  "TE-2-8 EV-2 Condenser Outlet Temp" %

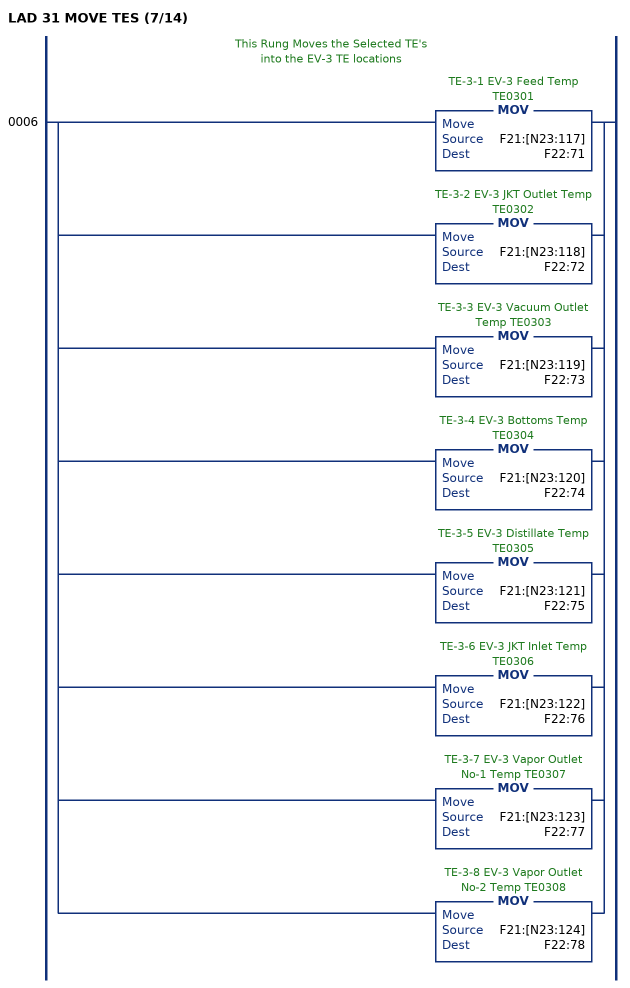
% Rung: 6 %
% This Rung Moves the Selected TE's
% into the EV-3 TE locations %
SOR BST MOV F21:[N23:117] F22:71 NXB MOV F21:[N23:118] F22:72 NXB MOV F21:[N23:119] F22:73 NXB MOV F21:[N23:120] F22:74 NXB MOV F21:[N23:121] F22:75 NXB MOV F21:[N23:122] F22:76 NXB MOV F21:[N23:123] F22:77 NXB MOV F21:[N23:124] F22:78 BND EOR
%   N23:117  TE0301_PTR  "TE-3-1 EV-3 Feed Temp PTR" %
%   F22:71  TE0301  "TE-3-1 EV-3 Feed Temp" %
%   N23:118  TE0302_PTR  "TE-3-2 EV-3 JKT Outlet Temp PTR" %
%   F22:72  TE0302  "TE-3-2 EV-3 JKT Outlet Temp" %
%   N23:119  TE0303_PTR  "TE-3-3 EV-3 Condenser Inlet Temp PTR" %
%   F22:73  TE0303  "TE-3-3 EV-3 Vacuum Outlet Temp" %
%   N23:120  TE0304_PTR  "TE-3-4 EV-3 Bottoms Temp PTR" %
%   F22:74  TE0304  "TE-3-4 EV-3 Bottoms Temp" %
%   N23:121  TE0305_PTR  "TE-3-5 EV-3 Distillate Temp PTR" %
%   F22:75  TE0305  "TE-3-5 EV-3 Distillate Temp" %
%   N23:122  TE0306_PTR  "TE-3-6 EV-3 JKT Inlet Temp PTR" %
%   F22:76  TE0306  "TE-3-6 EV-3 JKT Inlet Temp" %
%   N23:123  TE0307_PTR  "TE-3-7 EV-3 JKT Condensate Outlet Temp PTR" %
%   F22:77  TE0307  "TE-3-7 EV-3 Vapor Outlet No-1 Temp" %
%   N23:124  TE0308_PTR  "TE-3-8 EV-3 Condenser Outlet Temp PTR" %
%   F22:78  TE0308  "TE-3-8 EV-3 Vapor Outlet No-2 Temp" %

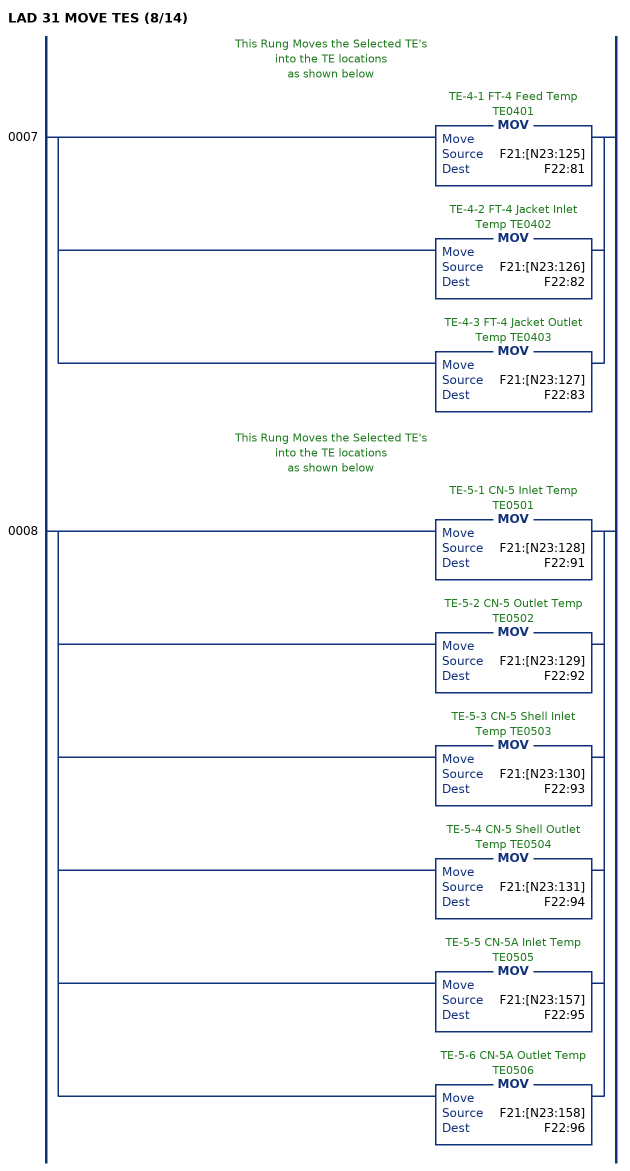
% Rung: 7 %
% This Rung Moves the Selected TE's
% into the TE locations
% as shown below %
SOR BST MOV F21:[N23:125] F22:81 NXB MOV F21:[N23:126] F22:82 NXB MOV F21:[N23:127] F22:83 BND EOR
%   N23:125  TE0401_PTR  "TE-4-1 FT-4 Feed Temp PTR" %
%   F22:81  TE0401  "TE-4-1 FT-4 Feed Temp" %
%   N23:126  TE0402_PTR  "TE-4-2 FT-4 Jacket Inlet Temp PTR" %
%   F22:82  TE0402  "TE-4-2 FT-4 Jacket Inlet Temp" %
%   N23:127  TE0403_PTR  "TE-4-3 FT-4 Jacket Outlet Temp PTR" %
%   F22:83  TE0403  "TE-4-3 FT-4 Jacket Outlet Temp" %
% Rung: 8 %
% This Rung Moves the Selected TE's
% into the TE locations
% as shown below %
SOR BST MOV F21:[N23:128] F22:91 NXB MOV F21:[N23:129] F22:92 NXB MOV F21:[N23:130] F22:93 NXB MOV F21:[N23:131] F22:94 NXB MOV F21:[N23:157] F22:95 NXB MOV F21:[N23:158] F22:96 BND EOR
%   N23:128  TE0501_PTR  "TE-5-1 CN-5 Inlet Temp PTR" %
%   F22:91  TE0501  "TE-5-1 CN-5 Inlet Temp" %
%   N23:129  TE0502_PTR  "TE-5-2 CN-5 Outlet Temp PTR" %
%   F22:92  TE0502  "TE-5-2 CN-5 Outlet Temp" %
%   N23:130  TE0503_PTR  "TE-5-3 CN-5 Shell Inlet Temp PTR" %
%   F22:93  TE0503  "TE-5-3 CN-5 Shell Inlet Temp" %
%   N23:131  TE0504_PTR  "TE-5-4 CN-5 Shell Outlet Temp PTR" %
%   F22:94  TE0504  "TE-5-4 CN-5 Shell Outlet Temp" %
%   N23:157  TE0505_PTR  "TE-5-1 CN-5A Inlet Temp PTR" %
%   F22:95  TE0505  "TE-5-5 CN-5A Inlet Temp" %
%   N23:158  TE0506_PTR  "TE-5-1 CN-5A Outlet Temp PTR" %
%   F22:96  TE0506  "TE-5-6 CN-5A Outlet Temp" %

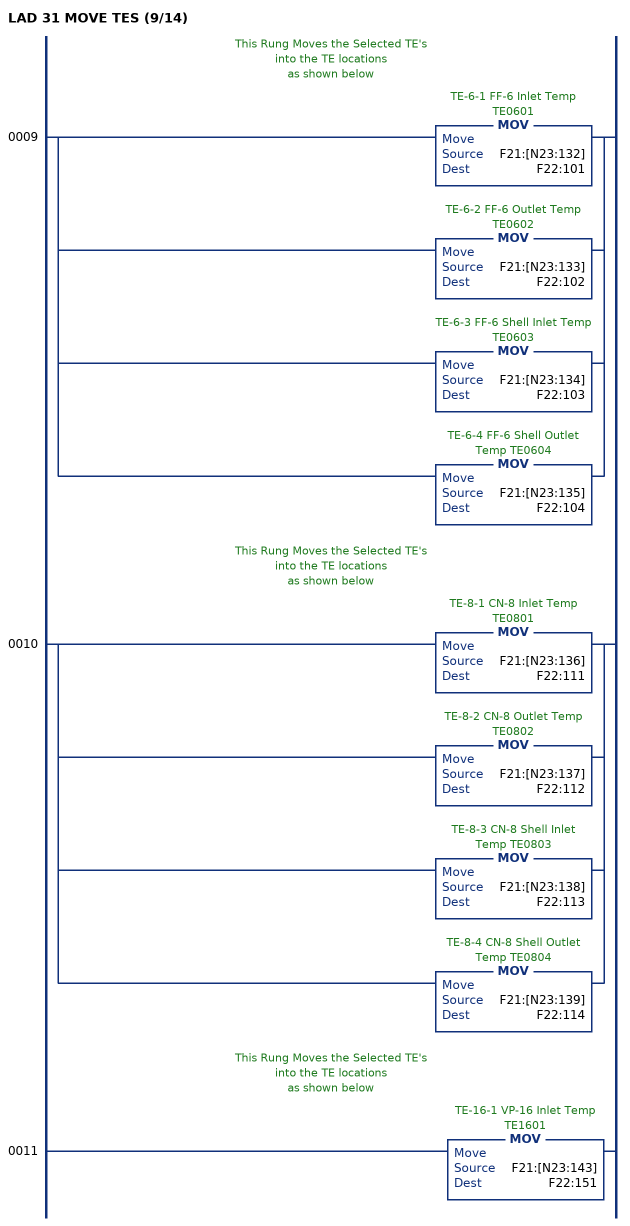
% Rung: 9 %
% This Rung Moves the Selected TE's
% into the TE locations
% as shown below %
SOR BST MOV F21:[N23:132] F22:101 NXB MOV F21:[N23:133] F22:102 NXB MOV F21:[N23:134] F22:103 NXB MOV F21:[N23:135] F22:104 BND EOR
%   N23:132  TE0601_PTR  "TE-6-1 FF-6 Inlet Temp PTR" %
%   F22:101  TE0601  "TE-6-1 FF-6 Inlet Temp" %
%   N23:133  TE0602_PTR  "TE-6-2 FF-6 Outlet Temp PTR" %
%   F22:102  TE0602  "TE-6-2 FF-6 Outlet Temp" %
%   N23:134  TE0603_PTR  "TE-6-3 FF-6 Shell Inlet Temp PTR" %
%   F22:103  TE0603  "TE-6-3 FF-6 Shell Inlet Temp" %
%   N23:135  TE0604_PTR  "TE-6-4 FF-6 Shell Outlet Temp PTR" %
%   F22:104  TE0604  "TE-6-4 FF-6 Shell Outlet Temp" %
% Rung: 10 %
% This Rung Moves the Selected TE's
% into the TE locations
% as shown below %
SOR BST MOV F21:[N23:136] F22:111 NXB MOV F21:[N23:137] F22:112 NXB MOV F21:[N23:138] F22:113 NXB MOV F21:[N23:139] F22:114 BND EOR
%   N23:136  TE0801_PTR  "TE-8-1 CN-8 Inlet Temp PTR" %
%   F22:111  TE0801  "TE-8-1 CN-8 Inlet Temp" %
%   N23:137  TE0802_PTR  "TE-8-2 CN-8 Outlet Temp PTR" %
%   F22:112  TE0802  "TE-8-2 CN-8 Outlet Temp" %
%   N23:138  TE0803_PTR  "TE-8-3 CN-8 Shell Inlet Temp PTR" %
%   F22:113  TE0803  "TE-8-3 CN-8 Shell Inlet Temp" %
%   N23:139  TE0804_PTR  "TE-8-4 CN-8 Shell Outlet Temp PTR" %
%   F22:114  TE0804  "TE-8-4 CN-8 Shell Outlet Temp" %
% Rung: 11 %
% This Rung Moves the Selected TE's
% into the TE locations
% as shown below %
SOR MOV F21:[N23:143] F22:151 EOR
%   N23:143  TE1601_PTR  "TE-16-1 VP-16 Inlet Temp PTR" %
%   F22:151  TE1601  "TE-16-1 VP-16 Inlet Temp" %

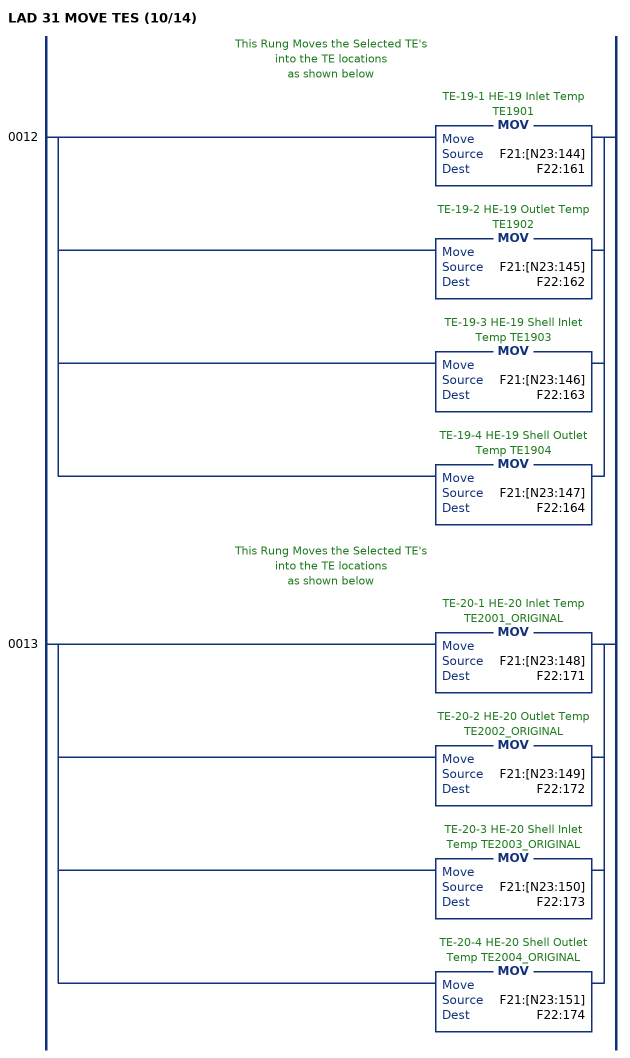
% Rung: 12 %
% This Rung Moves the Selected TE's
% into the TE locations
% as shown below %
SOR BST MOV F21:[N23:144] F22:161 NXB MOV F21:[N23:145] F22:162 NXB MOV F21:[N23:146] F22:163 NXB MOV F21:[N23:147] F22:164 BND EOR
%   N23:144  TE1901_PTR  "TE-19-1 HE-19 Inlet Temp PTR" %
%   F22:161  TE1901  "TE-19-1 HE-19 Inlet Temp" %
%   N23:145  TE1902_PTR  "TE-19-2 HE-19 Outlet Temp PTR" %
%   F22:162  TE1902  "TE-19-2 HE-19 Outlet Temp" %
%   N23:146  TE1903_PTR  "TE-19-3 HE-19 Shell Inlet Temp PTR" %
%   F22:163  TE1903  "TE-19-3 HE-19 Shell Inlet Temp" %
%   N23:147  TE1904_PTR  "TE-19-4 HE-19 Shell Outlet Temp PTR" %
%   F22:164  TE1904  "TE-19-4 HE-19 Shell Outlet Temp" %
% Rung: 13 %
% This Rung Moves the Selected TE's
% into the TE locations
% as shown below %
SOR BST MOV F21:[N23:148] F22:171 NXB MOV F21:[N23:149] F22:172 NXB MOV F21:[N23:150] F22:173 NXB MOV F21:[N23:151] F22:174 BND EOR
%   N23:148  TE2001_PTR_ORIGINAL  "TE-20-1 HE-20 Inlet Temp PTR" %
%   F22:171  TE2001_ORIGINAL  "TE-20-1 HE-20 Inlet Temp" %
%   N23:149  TE2002_PTR_ORIGINAL  "TE-20-2 HE-20 Outlet Temp PTR" %
%   F22:172  TE2002_ORIGINAL  "TE-20-2 HE-20 Outlet Temp" %
%   N23:150  TE2003_PTR_ORIGINAL  "TE-20-3 HE-20 Shell Inlet Temp PTR" %
%   F22:173  TE2003_ORIGINAL  "TE-20-3 HE-20 Shell Inlet Temp" %
%   N23:151  TE2004_PTR_ORIGINAL  "TE-20-4 HE-20 Shell Outlet Temp PTR" %
%   F22:174  TE2004_ORIGINAL  "TE-20-4 HE-20 Shell Outlet Temp" %

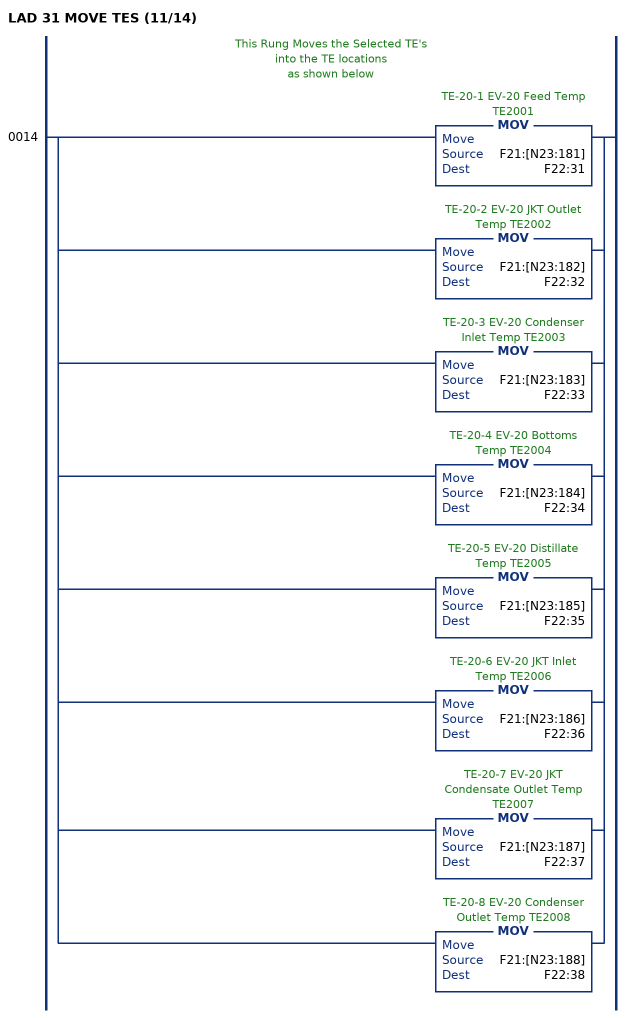
% Rung: 14 %
% This Rung Moves the Selected TE's
% into the TE locations
% as shown below %
SOR BST MOV F21:[N23:181] F22:31 NXB MOV F21:[N23:182] F22:32 NXB MOV F21:[N23:183] F22:33 NXB MOV F21:[N23:184] F22:34 NXB MOV F21:[N23:185] F22:35 NXB MOV F21:[N23:186] F22:36 NXB MOV F21:[N23:187] F22:37 NXB MOV F21:[N23:188] F22:38 BND EOR
%   N23:181  TE2001_PTR  "TE-20-1 Pointer" %
%   F22:31  TE2001  "TE-20-1 EV-20 Feed Temp" %
%   N23:182  TE2002_PTR  "TE-20-2 Pointer" %
%   F22:32  TE2002  "TE-20-2 EV-20 JKT Outlet Temp" %
%   N23:183  TE2003_PTR  "TE-20-3 Pointer" %
%   F22:33  TE2003  "TE-20-3 EV-20 Condenser Inlet Temp" %
%   N23:184  TE2004_PTR  "TE-20-4 Pointer" %
%   F22:34  TE2004  "TE-20-4 EV-20 Bottoms Temp" %
%   N23:185  TE2005_PTR  "TE-20-5 Pointer" %
%   F22:35  TE2005  "TE-20-5 EV-20 Distillate Temp" %
%   N23:186  TE2006_PTR  "TE-20-6 Pointer" %
%   F22:36  TE2006  "TE-20-6 EV-20 JKT Inlet Temp" %
%   N23:187  TE2007_PTR  "TE-20-7 Pointer" %
%   F22:37  TE2007  "TE-20-7 EV-20 JKT Condensate Outlet Temp" %
%   N23:188  TE2008_PTR  "TE-20-8 Pointer" %
%   F22:38  TE2008  "TE-20-8 EV-20 Condenser Outlet Temp" %

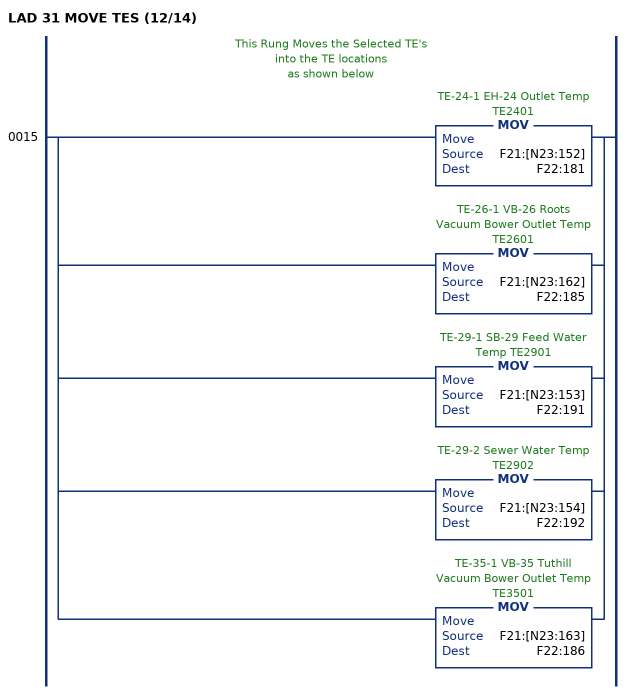
% Rung: 15 %
% This Rung Moves the Selected TE's
% into the TE locations
% as shown below %
SOR BST MOV F21:[N23:152] F22:181 NXB MOV F21:[N23:162] F22:185 NXB MOV F21:[N23:153] F22:191 NXB MOV F21:[N23:154] F22:192 NXB MOV F21:[N23:163] F22:186 BND EOR
%   N23:152  TE2401_PTR  "TE-24-1 EH-24 Outlet Temp PTR" %
%   F22:181  TE2401  "TE-24-1 EH-24 Outlet Temp" %
%   N23:162  TE2601_PTR  "TE-26-1 VB-26 Roots Vacuum Blower Disch Temp PTR" %
%   F22:185  TE2601  "TE-26-1 VB-26 Roots Vacuum Bower Outlet Temp" %
%   N23:153  TE2901_PTR  "TE-29-1 SB-29 Feed Water Temp PTR" %
%   F22:191  TE2901  "TE-29-1 SB-29 Feed Water Temp" %
%   N23:154  TE2902_PTR  "TE-29-2 Sewer Water Temp PTR" %
%   F22:192  TE2902  "TE-29-2 Sewer Water Temp" %
%   N23:163  TE3501_PTR  "TE-35-1 VB-35 Tuthill Vacuum Blower Disch Temp PTR" %
%   F22:186  TE3501  "TE-35-1 VB-35 Tuthill Vacuum Bower Outlet Temp" %

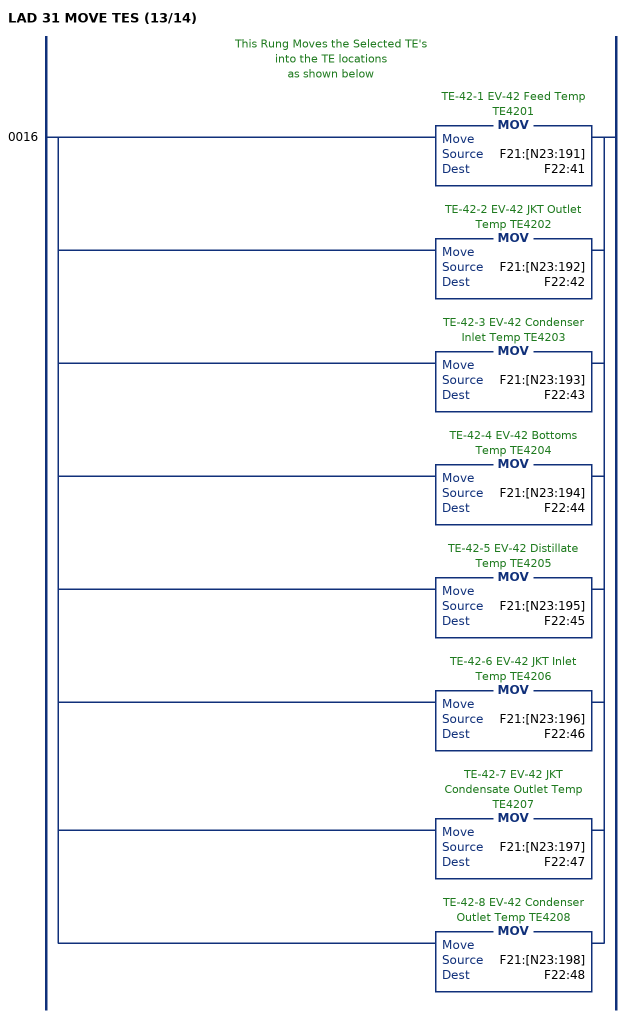
% Rung: 16 %
% This Rung Moves the Selected TE's
% into the TE locations
% as shown below %
SOR BST MOV F21:[N23:191] F22:41 NXB MOV F21:[N23:192] F22:42 NXB MOV F21:[N23:193] F22:43 NXB MOV F21:[N23:194] F22:44 NXB MOV F21:[N23:195] F22:45 NXB MOV F21:[N23:196] F22:46 NXB MOV F21:[N23:197] F22:47 NXB MOV F21:[N23:198] F22:48 BND EOR
%   N23:191  TE4201_PTR  "TE-42-1 Pointer" %
%   F22:41  TE4201  "TE-42-1 EV-42 Feed Temp" %
%   N23:192  TE4202_PTR  "TE-42-2 Pointer" %
%   F22:42  TE4202  "TE-42-2 EV-42 JKT Outlet Temp" %
%   N23:193  TE4203_PTR  "TE-42-3 Pointer" %
%   F22:43  TE4203  "TE-42-3 EV-42 Condenser Inlet Temp" %
%   N23:194  TE4204_PTR  "TE-42-4 Pointer" %
%   F22:44  TE4204  "TE-42-4 EV-42 Bottoms Temp" %
%   N23:195  TE4205_PTR  "TE-42-5 Pointer" %
%   F22:45  TE4205  "TE-42-5 EV-42 Distillate Temp" %
%   N23:196  TE4206_PTR  "TE-42-6 Pointer" %
%   F22:46  TE4206  "TE-42-6 EV-42 JKT Inlet Temp" %
%   N23:197  TE4207_PTR  "TE-42-7 Pointer" %
%   F22:47  TE4207  "TE-42-7 EV-42 JKT Condensate Outlet Temp" %
%   N23:198  TE4208_PTR  "TE-42-8 Pointer" %
%   F22:48  TE4208  "TE-42-8 EV-42 Condenser Outlet Temp" %

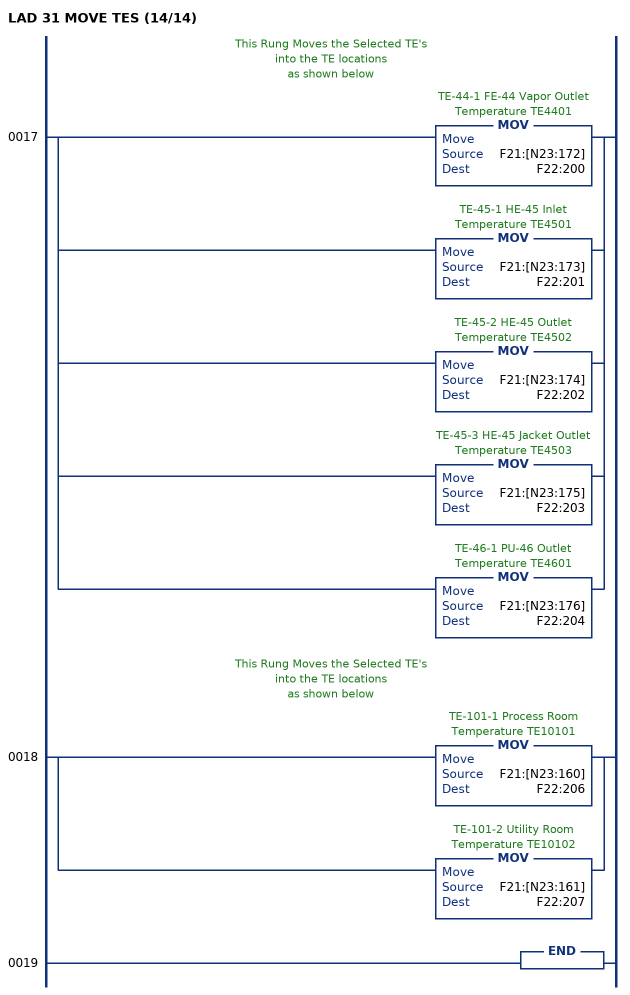
% Rung: 17 %
% This Rung Moves the Selected TE's
% into the TE locations
% as shown below %
SOR BST MOV F21:[N23:172] F22:200 NXB MOV F21:[N23:173] F22:201 NXB MOV F21:[N23:174] F22:202 NXB MOV F21:[N23:175] F22:203 NXB MOV F21:[N23:176] F22:204 BND EOR
%   N23:172  TE4401_PTR  "TE-44-1 FE-44 Vapor Outlet Temp PTR" %
%   F22:200  TE4401  "TE-44-1 FE-44 Vapor Outlet Temperature" %
%   N23:173  TE4501_PTR  "TE-45-1 HE-45 Inlet Temp PTR" %
%   F22:201  TE4501  "TE-45-1 HE-45 Inlet Temperature" %
%   N23:174  TE4502_PTR  "TE-45-1 HE-45 Outlet Temp PTR" %
%   F22:202  TE4502  "TE-45-2 HE-45 Outlet Temperature" %
%   N23:175  TE4503_PTR  "TE-45-1 HE-45 Jacket Outlet Temp PTR" %
%   F22:203  TE4503  "TE-45-3 HE-45 Jacket Outlet Temperature" %
%   N23:176  TE4601_PTR  "TE-46-1 PU-46 Outlet Temp PTR" %
%   F22:204  TE4601  "TE-46-1 PU-46 Outlet Temperature" %
% Rung: 18 %
% This Rung Moves the Selected TE's
% into the TE locations
% as shown below %
SOR BST MOV F21:[N23:160] F22:206 NXB MOV F21:[N23:161] F22:207 BND EOR
%   N23:160  TE10101_PTR  "TE-101-1 Process Room Temp PTR" %
%   F22:206  TE10101  "TE-101-1 Process Room Temperature" %
%   N23:161  TE10102_PTR  "TE-101-2 Utility Room Temp PTR" %
%   F22:207  TE10102  "TE-101-2 Utility Room Temperature" %
% Rung: 19 %
SOR END EOR

LADDER 32 "MOVE PTS"    % Move PT Info to Sequencial Locations, etc %
